RoboDK station: Stringer B Corner-Top-Long-BOX1.rdk

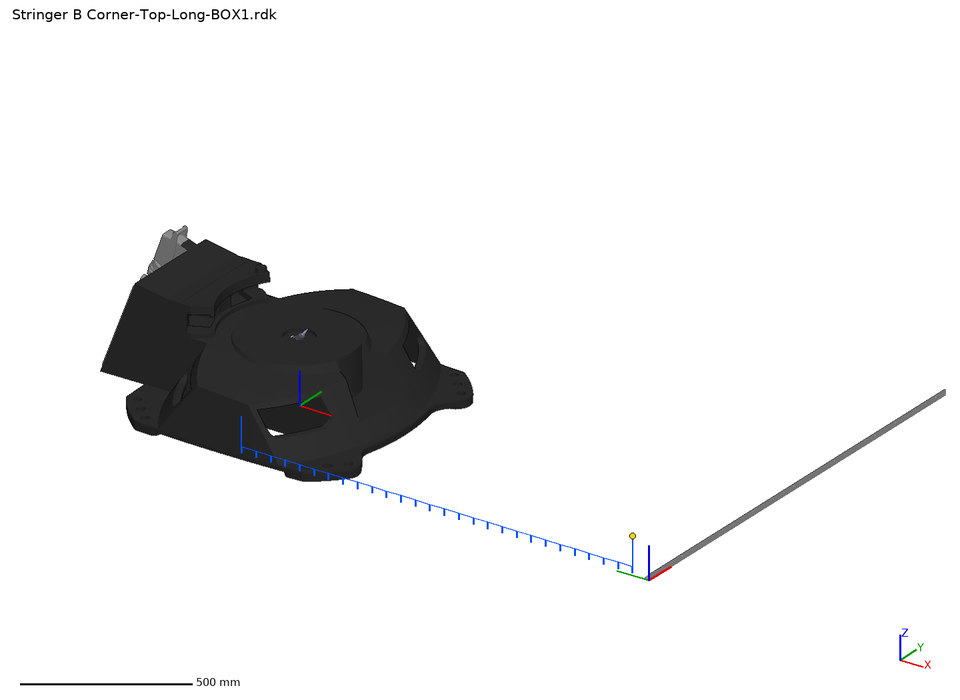
[picture v0: the station drawn from its stored meshes, robots at their saved joint values, targets as dots, program paths as lines]
Station Stringer B Corner-Top-Long-BOX1 (saved by RoboDK 5.2.3). Poses are relative to the parent item; angles as X-Y-Z fixed-axis rotations.
  - frame KUKA KR 210 R2700 extra Base at (0, 0, 0) mm
    - robot KUKA KR 210 R2700 extra: 6 axes, payload 210 kg, reach 2696 mm, repeatability 0.06 mm, weight 1068 kg
        joint limits [-185, -140, -120, -350, -125, -350] to [185, -5, 155, 350, 125, 350]; home [0, -90, 90, 0, 0, 0]; saved at [-34.328, -56.52, 112.84, -269.756, 20.787, 241.785]
      - tool Spindle, TCP at (32, 0, 260) mm, rotated rx 0 ry 39 rz 0 deg, size 157.3 x 72 x 259.9 mm
  - frame Frame 2 at (1618.38, -541.41, 103.58) mm, rotated rx 0 ry 0 rz 90 deg
    - object L-Stringer C-top-corner at (0, 0, 0) mm, size 1499.5 x 20 x 20 mm, geometry from L-Stringer C-top-corner.stl
    - object Stringer C-Corner-Top-Long-BOX1 at (0, 22.5, 0) mm, rotated rx 0 ry 0 rz -90 deg, 28 curves, geometry from Point 28
  - machining project Point settings: rotZ(0) | rotX(0)*rotY(0) | rotz(0) | onStart | onPathStart | onApproach | onPoint | onRetract | onFinish | SetRPM(%1) | SetTool(%1) | Extruder(%1) | default | default | OutOnMov(%1) | OutOffMov(%1) | onPathFinish | M_RunCode(%1) | 潫險潫險潫險潫險潫險潫險潫險潫險潫險潫險潫險潫險潫險潫險潫險潫險潫險潫險潫險潫險潫險潫險潫險潫險潫險潫險潫險潫險潫險潫險潫險潫險潫險潫險潫險潫險潫險潫險潫險潫險潫險潫險潫
  - program Point (151 instructions, listed below)
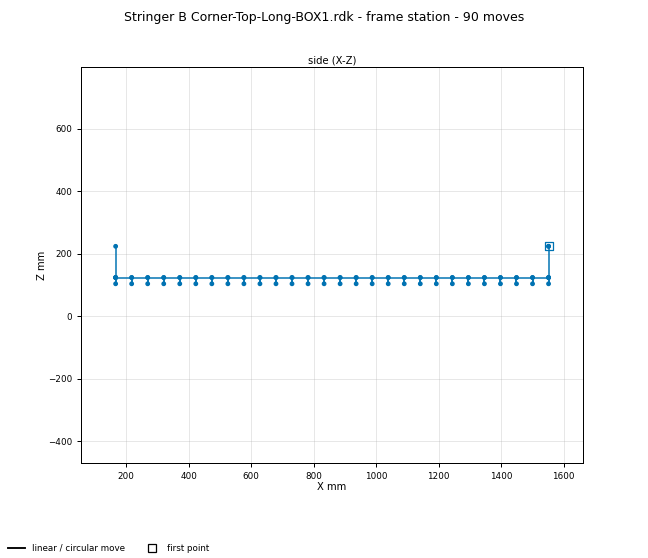
[picture p0: tool path of Stringer B Corner-Top-Long-BOX1.rdk in frame station, 90 of 90 moves have a stored position in this frame; points joined in program order, loops and branches not executed]

--- program Point (robot KUKA KR 210 R2700 extra) ---
  Smooth(1)
  Set speed (1000.0 mm/s)
  Set Ref.: Frame 2
  Set Tool: Spindle
  Show Spindle
  MoveJ 1 to (12.5, 66.57, 120) mm, rotated rx 180 ry 0 rz -180 deg; joints [19.589, -62.091, 124.046, -126.809, 15.28, 143.263]
  MoveL 2 to (12.5, 66.57, 120) mm, rotated rx 180 ry 0 rz -180 deg; joints [19.589, -62.091, 124.046, -126.809, 15.28, 143.263]
  MoveL 3 to (12.5, 66.57, 20) mm, rotated rx -180 ry 0 rz -180 deg; joints [19.589, -56.463, 123.473, -138.946, 18.739, 155.945]
  MoveL 4 to (12.5, 66.57, 20) mm, rotated rx -180 ry 0 rz -180 deg; joints [19.589, -56.463, 123.473, -138.946, 18.739, 155.945]
  Set speed (50.0 mm/s)
  MoveL 5 to (12.5, 66.57, 0) mm, rotated rx 180 ry 0 rz -180 deg; joints [19.589, -55.32, 123.298, -140.75, 19.48, 157.853]
  MoveL 6 to (12.5, 66.57, 20) mm, rotated rx -180 ry 0 rz -180 deg; joints [19.589, -56.463, 123.473, -138.946, 18.739, 155.945]
  Set speed (1000.0 mm/s)
  MoveL 7 to (12.5, 117.91, 20) mm, rotated rx 180 ry 0 rz 180 deg; joints [17.609, -56.821, 124.36, -143.515, 18.674, 158.84]
  Set speed (50.0 mm/s)
  MoveL 8 to (12.5, 117.91, 0) mm, rotated rx 180 ry 0 rz -180 deg; joints [17.609, -55.66, 124.183, -145.173, 19.473, 160.595]
  MoveL 9 to (12.5, 117.91, 20) mm, rotated rx 180 ry 0 rz 180 deg; joints [17.609, -56.821, 124.36, -143.515, 18.674, 158.84]
  Set speed (1000.0 mm/s)
  MoveL 10 to (12.5, 169.24, 20) mm, rotated rx 180 ry 0 rz 180 deg; joints [15.585, -57.136, 125.152, -148.056, 18.637, 161.655]
  Set speed (50.0 mm/s)
  MoveL 11 to (12.5, 169.24, 0) mm, rotated rx 180 ry 0 rz 180 deg; joints [15.585, -55.96, 124.973, -149.551, 19.49, 163.237]
  MoveL 12 to (12.5, 169.24, 20) mm, rotated rx 180 ry 0 rz 180 deg; joints [15.585, -57.136, 125.152, -148.056, 18.637, 161.655]
  Set speed (1000.0 mm/s)
  MoveL 13 to (12.5, 220.57, 20) mm, rotated rx -180 ry 0 rz -180 deg; joints [13.52, -57.411, 125.845, -152.563, 18.621, 164.388]
  Set speed (50.0 mm/s)
  MoveL 14 to (12.5, 220.57, 0) mm, rotated rx -180 ry 0 rz 180 deg; joints [13.52, -56.22, 125.665, -153.879, 19.523, 165.78]
  MoveL 15 to (12.5, 220.57, 20) mm, rotated rx -180 ry 0 rz -180 deg; joints [13.52, -57.411, 125.845, -152.563, 18.621, 164.388]
  Set speed (1000.0 mm/s)
  MoveL 16 to (12.5, 271.91, 20) mm, rotated rx -180 ry 0 rz -180 deg; joints [11.419, -57.644, 126.44, -157.034, 18.622, 167.041]
  Set speed (50.0 mm/s)
  MoveL 17 to (12.5, 271.91, 0) mm, rotated rx 180 ry 0 rz 180 deg; joints [11.419, -56.442, 126.258, -158.158, 19.565, 168.23]
  MoveL 18 to (12.5, 271.91, 20) mm, rotated rx -180 ry 0 rz -180 deg; joints [11.419, -57.644, 126.44, -157.034, 18.622, 167.041]
  Set speed (1000.0 mm/s)
  MoveL 19 to (12.5, 323.24, 20) mm, rotated rx 180 ry 0 rz 180 deg; joints [9.286, -57.837, 126.933, -161.466, 18.632, 169.618]
  Set speed (50.0 mm/s)
  MoveL 20 to (12.5, 323.24, 0) mm, rotated rx 180 ry 0 rz -180 deg; joints [9.286, -56.624, 126.75, -162.388, 19.611, 170.593]
  MoveL 21 to (12.5, 323.24, 20) mm, rotated rx 180 ry 0 rz 180 deg; joints [9.286, -57.837, 126.933, -161.466, 18.632, 169.618]
  Set speed (1000.0 mm/s)
  MoveL 22 to (12.5, 374.57, 20) mm, rotated rx 180 ry 0 rz -180 deg; joints [7.127, -57.989, 127.324, -165.864, 18.646, 172.129]
  Set speed (50.0 mm/s)
  MoveL 23 to (12.5, 374.57, 0) mm, rotated rx -180 ry 0 rz -180 deg; joints [7.127, -56.767, 127.14, -166.575, 19.653, 172.882]
  MoveL 24 to (12.5, 374.57, 20) mm, rotated rx 180 ry 0 rz -180 deg; joints [7.127, -57.989, 127.324, -165.864, 18.646, 172.129]
  Set speed (1000.0 mm/s)
  MoveL 25 to (12.5, 425.91, 20) mm, rotated rx 180 ry 0 rz 180 deg; joints [4.947, -58.1, 127.612, -170.234, 18.66, 174.586]
  Set speed (50.0 mm/s)
  MoveL 26 to (12.5, 425.91, 0) mm, rotated rx 180 ry 0 rz 180 deg; joints [4.947, -56.872, 127.427, -170.729, 19.688, 175.111]
  MoveL 27 to (12.5, 425.91, 20) mm, rotated rx 180 ry 0 rz 180 deg; joints [4.947, -58.1, 127.612, -170.234, 18.66, 174.586]
  Set speed (1000.0 mm/s)
  MoveL 28 to (12.5, 477.24, 20) mm, rotated rx -180 ry 0 rz -180 deg; joints [2.754, -58.17, 127.796, -174.581, 18.671, 177.005]
  Set speed (50.0 mm/s)
  MoveL 29 to (12.5, 477.24, 0) mm, rotated rx -180 ry 0 rz -180 deg; joints [2.754, -56.939, 127.61, -174.858, 19.712, 177.298]
  MoveL 30 to (12.5, 477.24, 20) mm, rotated rx -180 ry 0 rz -180 deg; joints [2.754, -58.17, 127.796, -174.581, 18.671, 177.005]
  Set speed (1000.0 mm/s)
  MoveL 31 to (12.5, 528.57, 20) mm, rotated rx -180 ry 0 rz -180 deg; joints [0.552, -58.201, 127.874, -178.916, 18.675, 179.402]
  Set speed (50.0 mm/s)
  MoveL 32 to (12.5, 528.57, 0) mm, rotated rx -180 ry 0 rz -180 deg; joints [0.552, -56.967, 127.689, -178.971, 19.723, 179.46]
  MoveL 33 to (12.5, 528.57, 20) mm, rotated rx -180 ry 0 rz -180 deg; joints [0.552, -58.201, 127.874, -178.916, 18.675, 179.402]
  Set speed (1000.0 mm/s)
  MoveL 34 to (12.5, 579.91, 20) mm, rotated rx 180 ry 0 rz -180 deg; joints [-1.653, -58.191, 127.848, -183.249, 18.674, 181.794]
  Set speed (50.0 mm/s)
  MoveL 35 to (12.5, 579.91, 0) mm, rotated rx 180 ry 0 rz 180 deg; joints [-1.653, -56.958, 127.662, -183.083, 19.719, 181.618]
  MoveL 36 to (12.5, 579.91, 20) mm, rotated rx 180 ry 0 rz -180 deg; joints [-1.653, -58.191, 127.848, -183.249, 18.674, 181.794]
  Set speed (1000.0 mm/s)
  MoveL 37 to (12.5, 631.24, 20) mm, rotated rx 180 ry 0 rz 180 deg; joints [-3.851, -58.14, 127.717, -187.589, 18.666, 184.2]
  Set speed (50.0 mm/s)
  MoveL 38 to (12.5, 631.24, 0) mm, rotated rx 180 ry 0 rz -180 deg; joints [-3.851, -56.91, 127.532, -187.203, 19.702, 183.79]
  MoveL 39 to (12.5, 631.24, 20) mm, rotated rx 180 ry 0 rz 180 deg; joints [-3.851, -58.14, 127.717, -187.589, 18.666, 184.2]
  Set speed (1000.0 mm/s)
  MoveL 40 to (12.5, 682.57, 20) mm, rotated rx -180 ry 0 rz -180 deg; joints [-6.039, -58.049, 127.481, -191.946, 18.653, 186.636]
  Set speed (50.0 mm/s)
  MoveL 41 to (12.5, 682.57, 0) mm, rotated rx -180 ry 0 rz -180 deg; joints [-6.039, -56.824, 127.297, -191.342, 19.672, 185.996]
  MoveL 42 to (12.5, 682.57, 20) mm, rotated rx -180 ry 0 rz -180 deg; joints [-6.039, -58.049, 127.481, -191.946, 18.653, 186.636]
  Set speed (1000.0 mm/s)
  MoveL 43 to (12.5, 733.91, 20) mm, rotated rx 180 ry 0 rz -180 deg; joints [-8.209, -57.918, 127.142, -196.33, 18.638, 189.119]
  Set speed (50.0 mm/s)
  MoveL 44 to (12.5, 733.91, 0) mm, rotated rx 180 ry 0 rz 180 deg; joints [-8.209, -56.7, 126.958, -195.512, 19.632, 188.254]
  MoveL 45 to (12.5, 733.91, 20) mm, rotated rx 180 ry 0 rz -180 deg; joints [-8.209, -57.918, 127.142, -196.33, 18.638, 189.119]
  Set speed (1000.0 mm/s)
  MoveL 46 to (12.5, 785.24, 20) mm, rotated rx 180 ry 0 rz 180 deg; joints [-10.356, -57.746, 126.699, -200.744, 18.626, 191.661]
  Set speed (50.0 mm/s)
  MoveL 47 to (12.5, 785.24, 0) mm, rotated rx -180 ry 0 rz -180 deg; joints [-10.356, -56.538, 126.517, -199.72, 19.588, 190.578]
  MoveL 48 to (12.5, 785.24, 20) mm, rotated rx 180 ry 0 rz 180 deg; joints [-10.356, -57.746, 126.699, -200.744, 18.626, 191.661]
  Set speed (1000.0 mm/s)
  MoveL 49 to (12.5, 836.57, 20) mm, rotated rx 180 ry 0 rz -180 deg; joints [-12.473, -57.533, 126.155, -205.195, 18.62, 194.275]
  Set speed (50.0 mm/s)
  MoveL 50 to (12.5, 836.57, 0) mm, rotated rx 180 ry 0 rz -180 deg; joints [-12.473, -56.336, 125.974, -203.974, 19.543, 192.983]
  MoveL 51 to (12.5, 836.57, 20) mm, rotated rx 180 ry 0 rz -180 deg; joints [-12.473, -57.533, 126.155, -205.195, 18.62, 194.275]
  Set speed (1000.0 mm/s)
  MoveL 52 to (12.5, 887.91, 20) mm, rotated rx -180 ry 0 rz -180 deg; joints [-14.557, -57.279, 125.511, -209.685, 18.627, 196.967]
  Set speed (50.0 mm/s)
  MoveL 53 to (12.5, 887.91, 0) mm, rotated rx 180 ry 0 rz -180 deg; joints [-14.557, -56.095, 125.331, -208.277, 19.505, 195.478]
  MoveL 54 to (12.5, 887.91, 20) mm, rotated rx -180 ry 0 rz -180 deg; joints [-14.557, -57.279, 125.511, -209.685, 18.627, 196.967]
  Set speed (1000.0 mm/s)
  MoveL 55 to (12.5, 939.24, 20) mm, rotated rx 180 ry 0 rz 180 deg; joints [-16.602, -56.984, 124.768, -214.209, 18.652, 199.741]
  Set speed (50.0 mm/s)
  MoveL 56 to (12.5, 939.24, 0) mm, rotated rx -180 ry 0 rz -180 deg; joints [-16.602, -55.815, 124.59, -212.631, 19.479, 198.071]
  MoveL 57 to (12.5, 939.24, 20) mm, rotated rx 180 ry 0 rz 180 deg; joints [-16.602, -56.984, 124.768, -214.209, 18.652, 199.741]
  Set speed (1000.0 mm/s)
  MoveL 58 to (12.5, 990.57, 20) mm, rotated rx 180 ry 0 rz 180 deg; joints [-18.604, -56.647, 123.929, -218.765, 18.703, 202.597]
  Set speed (50.0 mm/s)
  MoveL 59 to (12.5, 990.57, 0) mm, rotated rx -180 ry 0 rz -180 deg; joints [-18.604, -55.495, 123.753, -217.032, 19.473, 200.763]
  MoveL 60 to (12.5, 990.57, 20) mm, rotated rx 180 ry 0 rz 180 deg; joints [-18.604, -56.647, 123.929, -218.765, 18.703, 202.597]
  Set speed (1000.0 mm/s)
  MoveL 61 to (12.5, 1041.91, 20) mm, rotated rx 180 ry 0 rz 180 deg; joints [-20.561, -56.27, 122.994, -223.343, 18.785, 205.529]
  Set speed (50.0 mm/s)
  MoveL 62 to (12.5, 1041.91, 0) mm, rotated rx 180 ry 0 rz -180 deg; joints [-20.561, -55.135, 122.82, -221.475, 19.494, 203.552]
  MoveL 63 to (12.5, 1041.91, 20) mm, rotated rx 180 ry 0 rz 180 deg; joints [-20.561, -56.27, 122.994, -223.343, 18.785, 205.529]
  Set speed (1000.0 mm/s)
  MoveL 64 to (12.5, 1093.24, 20) mm, rotated rx 180 ry 0 rz 180 deg; joints [-22.468, -55.85, 121.967, -227.928, 18.905, 208.527]
  Set speed (50.0 mm/s)
  MoveL 65 to (12.5, 1093.24, 0) mm, rotated rx 180 ry 0 rz 180 deg; joints [-22.468, -54.734, 121.795, -225.949, 19.55, 206.431]
  MoveL 66 to (12.5, 1093.24, 20) mm, rotated rx 180 ry 0 rz 180 deg; joints [-22.468, -55.85, 121.967, -227.928, 18.905, 208.527]
  Set speed (1000.0 mm/s)
  MoveL 67 to (12.5, 1144.57, 20) mm, rotated rx -180 ry 0 rz -180 deg; joints [-24.325, -55.39, 120.849, -232.506, 19.069, 211.577]
  Set speed (50.0 mm/s)
  MoveL 68 to (12.5, 1144.57, 0) mm, rotated rx -180 ry 0 rz -180 deg; joints [-24.325, -54.293, 120.679, -230.441, 19.647, 209.389]
  MoveL 69 to (12.5, 1144.57, 20) mm, rotated rx -180 ry 0 rz -180 deg; joints [-24.325, -55.39, 120.849, -232.506, 19.069, 211.577]
  Set speed (1000.0 mm/s)
  MoveL 70 to (12.5, 1195.91, 20) mm, rotated rx 180 ry 0 rz -180 deg; joints [-26.128, -54.888, 119.641, -237.059, 19.283, 214.665]
  Set speed (50.0 mm/s)
  MoveL 71 to (12.5, 1195.91, 0) mm, rotated rx -180 ry 0 rz -180 deg; joints [-26.128, -53.81, 119.474, -234.933, 19.792, 212.41]
  MoveL 72 to (12.5, 1195.91, 20) mm, rotated rx 180 ry 0 rz -180 deg; joints [-26.128, -54.888, 119.641, -237.059, 19.283, 214.665]
  Set speed (1000.0 mm/s)
  MoveL 73 to (12.5, 1247.24, 20) mm, rotated rx 180 ry 0 rz -180 deg; joints [-27.878, -54.344, 118.347, -241.564, 19.55, 217.769]
  Set speed (50.0 mm/s)
  MoveL 74 to (12.5, 1247.24, 0) mm, rotated rx -180 ry 0 rz -180 deg; joints [-27.878, -53.287, 118.181, -239.405, 19.99, 215.476]
  MoveL 75 to (12.5, 1247.24, 20) mm, rotated rx 180 ry 0 rz -180 deg; joints [-27.878, -54.344, 118.347, -241.564, 19.55, 217.769]
  Set speed (1000.0 mm/s)
  MoveL 76 to (12.5, 1298.57, 20) mm, rotated rx 180 ry 0 rz -180 deg; joints [-29.573, -53.759, 116.967, -246.002, 19.875, 220.871]
  Set speed (50.0 mm/s)
  MoveL 77 to (12.5, 1298.57, 0) mm, rotated rx 180 ry 0 rz 180 deg; joints [-29.573, -52.723, 116.804, -243.837, 20.245, 218.566]
  MoveL 78 to (12.5, 1298.57, 20) mm, rotated rx 180 ry 0 rz -180 deg; joints [-29.573, -53.759, 116.967, -246.002, 19.875, 220.871]
  Set speed (1000.0 mm/s)
  MoveL 79 to (12.5, 1349.91, 20) mm, rotated rx 180 ry 0 rz 180 deg; joints [-31.213, -53.133, 115.502, -250.352, 20.26, 223.949]
  Set speed (50.0 mm/s)
  MoveL 80 to (12.5, 1349.91, 0) mm, rotated rx 180 ry 0 rz -180 deg; joints [-31.213, -52.118, 115.342, -248.205, 20.563, 221.659]
  MoveL 81 to (12.5, 1349.91, 20) mm, rotated rx 180 ry 0 rz 180 deg; joints [-31.213, -53.133, 115.502, -250.352, 20.26, 223.949]
  Set speed (1000.0 mm/s)
  MoveL 82 to (12.5, 1401.24, 20) mm, rotated rx 180 ry 0 rz 180 deg; joints [-32.797, -52.465, 113.956, -254.595, 20.707, 226.985]
  Set speed (50.0 mm/s)
  MoveL 83 to (12.5, 1401.24, 0) mm, rotated rx 180 ry 0 rz -180 deg; joints [-32.797, -51.471, 113.797, -252.489, 20.944, 224.732]
  MoveL 84 to (12.5, 1401.24, 20) mm, rotated rx 180 ry 0 rz 180 deg; joints [-32.797, -52.465, 113.956, -254.595, 20.707, 226.985]
  Set speed (1000.0 mm/s)
  MoveL 85 to (12.5, 1452.57, 20) mm, rotated rx -180 ry 0 rz -180 deg; joints [-34.328, -51.756, 112.329, -258.713, 21.216, 229.962]
  Set speed (50.0 mm/s)
  MoveL 86 to (12.5, 1452.57, 0) mm, rotated rx 180 ry 0 rz 180 deg; joints [-34.328, -50.783, 112.172, -256.668, 21.39, 227.766]
  MoveL 87 to (12.5, 1452.57, 20) mm, rotated rx -180 ry 0 rz -180 deg; joints [-34.328, -51.756, 112.329, -258.713, 21.216, 229.962]
  MoveL 88 to (12.5, 1452.57, 20) mm, rotated rx -180 ry 0 rz -180 deg; joints [-34.328, -51.756, 112.329, -258.713, 21.216, 229.962]
  Set speed (1000.0 mm/s)
  MoveL 89 to (12.5, 1452.57, 20) mm, rotated rx -180 ry 0 rz -180 deg; joints [-34.328, -51.756, 112.329, -258.713, 21.216, 229.962]
  MoveL 90 to (12.5, 1452.57, 120) mm, rotated rx 180 ry 0 rz 180 deg; joints [-34.328, -56.52, 112.84, -269.756, 20.787, 241.785]
